// TIA Portal V18 export
DATA_BLOCK "Control_Buttons_Manipulate_DB"   // DB90
VERSION : 0.1
// stored: AutoNumber true, DBAccessibleFromOPCUA true, InstanceOfName Control_Buttons_Manipulate, InstanceOfType FB
"Control_Buttons_Manipulate"
   // VAR_INPUT
   //    JogInZ1pos : Bool;
   //    JogInZ1neg : Bool;
   //    JogInZ2pos : Bool;
   //    JogInZ2neg : Bool;
   //    InXhome : Bool;
   //    InYhome : Bool;
   //    InZ1home : Bool;
   //    InZ2home : Bool;
   //    MovePermission : Bool;
   //    ReadyDevices : Bool;
   // END_VAR
   // VAR_OUTPUT
   //    JogOutXpos : Bool;
   //    JogOutXneg : Bool;
   //    JogOutYpos : Bool;
   //    JogOutYneg : Bool;
   //    JogOutZ1pos : Bool;
   //    JogOutZ1neg : Bool;
   //    JogOutZ2pos : Bool;
   //    JogOutZ2neg : Bool;
   //    XHoming : Bool;
   //    YHoming : Bool;
   //    Z1Homing : Bool;
   //    Z2Homing : Bool;
   //    StartMachine : Bool;
   // END_VAR
   // VAR
   //    ButtonsReadyToRead : Bool;
   //    XYmoveout : Bool;
   // END_VAR
BEGIN
END_DATA_BLOCK
